(* CoDeSys 2.3.9.35 project: SISTEMA_2_SEMAFOROS.pro *)
(* Author: Franklin *)
(* Libraries: SysLibTargetVisu.lib 26.11.08 09:50:36, Standard.lib 26.11.08 09:46:20, Iecsfc.lib 26.11.08 09:46:14, DU35x.lib 26.11.09 14:36:14, SYSLIBCALLBACK.LIB 26.11.08 09:50:38 *)

(* PLC configuration (modules and I/O channels)
PLC Configuration [Root] node -1, in %IB0 out %QB0
  Communication [Comunica] node 0, in %IB0 out %QB0
    COM1 [COM1] node 0, in %IB0 out %QB0 {BaudRate = 115200; Paridade = No Parity; StopBits = 1 Stop Bit; Modem = Without RTS/CTS; Delay = 5}
      MToolIEC [Codesys] node 0, in %IB0 out %QB0
    COM2 [COM2] node 1, in %IB0 out %QB0 {BaudRate = 115200; Paridade = No Parity; StopBits = 1 Stop Bit; Modem = Without RTS/CTS; Delay = 5}
      Disable [Desabilitado485] node 0, in %IB0 out %QB0
  Bus [Barramento] node 1, in %IB0 out %QB0
    Inputs [Entradas] node 0, in %IB0 out %QB0
      Digital Inputs 0 [Entradas0] node 0, in %IW0 out %QB0
        I00 AT %IX0.0 [BitInput] I0.0
        I01 AT %IX0.1 [BitInput] I0.1
        I02 AT %IX0.2 [BitInput] I0.2
        I03 AT %IX0.3 [BitInput] I0.3
        I04 AT %IX0.4 [BitInput] I0.4
        I05 AT %IX0.5 [BitInput] I0.5
        I06 AT %IX0.6 [BitInput] I0.6
        I07 AT %IX0.7 [BitInput] I0.7
        I08 AT %IX0.8 [BitInput] I0.8
      Digital Inputs 1 [Entradas1] node 0, in %IW1 out %QB0
        I10 AT %IX1.0 [BitInput] I1.0
        I11 AT %IX1.1 [BitInput] I1.1
        I12 AT %IX1.2 [BitInput] I1.2
        I13 AT %IX1.3 [BitInput] I1.3
        I14 AT %IX1.4 [BitInput] I1.4
        I15 AT %IX1.5 [BitInput] I1.5
        I16 AT %IX1.6 [BitInput] I1.6
        I17 AT %IX1.7 [BitInput] I1.7
        I18 AT %IX1.8 [BitInput] I1.8
      Digital Inputs 2 [Entradas2] node 0, in %IW2 out %QB0
        I20 AT %IX2.0 [BitInput] I2.0
        I21 AT %IX2.1 [BitInput] I2.1
      Analog Inputs [EntradaAnalogica] node 0, in %IW4 out %QB0
        AI0 AT %IW4 [WordInput] AI0 {TipoAnalogica = Channel Disable; FiltroAnalogica = Filter 0 - AI=2ms  / AV=90ms; FundoEscala = 0}
        AI1 AT %IW5 [WordInput] AI1 {TipoAnalogica = Channel Disable; FiltroAnalogica = Filter 0 - AI=2ms  / AV=90ms; FundoEscala = 0}
        AI2 AT %IW6 [WordInput] AI2 {TipoAnalogica = Channel Disable; FiltroAnalogica = Filter 0 - AI=2ms  / AV=90ms; FundoEscala = 0}
        AI3 AT %IW7 [WordInput] AI3 {TipoAnalogica = Channel Disable; FiltroAnalogica = Filter 0 - AI=2ms  / AV=90ms; FundoEscala = 0}
      Fast Inputs [EntradasRapidas] node 1, in %IB16 out %QB0
        Block 0 [Bloco0] node 0, in %IB16 out %QB0
          Disable [DesabilitadoBloco0] node 0, in %IB16 out %QB0
        Block 1 [Bloco1] node 1, in %IB16 out %QB0
          Disable [DesabilitadoBloco1] node 0, in %IB16 out %QB0
        Configurable Input Block 0 [EntradaConfiBloco0] node 2, in %IB16 out %QB0
          Counter 0 [EntradaConfContador0] node 0, in %IB16 out %QB0 {EntradaConfiguravelContador = Disable}
        Configurable Input Block 1 [EntradaConfiBloco1] node 3, in %IB16 out %QB0
          Counter 2 [EntradaConfContador2] node 0, in %IB16 out %QB0 {EntradaConfiguravelContador = Disable}
    Outputs [Saidas] node 1, in %IB13 out %QB0
      Digital Outputs 0 [Saidas0] node 0, in %IW0 out %QW0
        Q00 AT %QX0.0 [BitOutput] Q0.0
        Q01 AT %QX0.1 [BitOutput] Q0.1
        Q02 AT %QX0.2 [BitOutput] Q0.2
        Q03 AT %QX0.3 [BitOutput] Q0.3
        Q04 AT %QX0.4 [BitOutput] Q0.4
        Q05 AT %QX0.5 [BitOutput] Q0.5
        Q06 AT %QX0.6 [BitOutput] Q0.6
        Q07 AT %QX0.7 [BitOutput] Q0.7
      Digital Outputs 1 [Saidas1] node 0, in %IW0 out %QW1
        Q10 AT %QX1.0 [BitOutput] Q1.0
        Q11 AT %QX1.1 [BitOutput] Q1.1
        Q12 AT %QX1.2 [BitOutput] Q1.2
        Q13 AT %QX1.3 [BitOutput] Q1.3
        Q14 AT %QX1.4 [BitOutput] Q1.4
        Q15 AT %QX1.5 [BitOutput] Q1.5
        Q16 AT %QX1.6 [BitOutput] Q1.6
        Q17 AT %QX1.7 [BitOutput] Q1.7
      Analog Outputs [SaidaAnalogica] node 0, in %IW0 out %QW3
        AO0 AT %QW3 [WordOutput] AO0 {TipoAnalogica = Channel Disable; FundoEscala = 0}
        AO1 AT %QW4 [WordOutput] AO1 {TipoAnalogica = Channel Disable; FundoEscala = 0}
      Fast Outputs [SaidasRapidas] node 1, in %IB0 out %QB10
        Fast Output 0 Disable [DesabilitadoF0] node 0, in %IB0 out %QB10
        Fast Output 1 Disable [DesabilitadoF1] node 1, in %IB0 out %QB10
      Counter Output [SaidasContador] node 2, in %IB0 out %QB10
        Block 0 Output Disable [DesabilitadoSaidaBloco0] node 0, in %IB0 out %QB10
        Block 1 Output Disable [DesabilitadoSaidaBloco1] node 1, in %IB0 out %QB10
  External Events [Eventos] node 2, in %IB13 out %QB6
    Timer Event [TimerEvent] node 0, in %IB13 out %QB6 {Intervalo = 10}
*)

(* POU PLC_PRG, LD *)
PROGRAM PLC_PRG
(*
	 autor; franklin
	 descricao: codigo estruturado com base em um autômato finito determinísco (AFD) para controle de maquina de estados finita
*)

VAR
	botao AT %IX0.0: BOOL;
	S0 AT %MX0.0: BOOL;
	T1: TON;
	A_VERDE AT %QX1.2: BOOL;
	B_VERMELHO AT %QX1.3: BOOL;
	S1 AT %MX0.1: BOOL;
	botao_pulso: R_TRIG;
	A_AMARELO AT %QX1.1: BOOL;
	T2: TON;
	S2 AT %MX0.2: BOOL;
	B_VERDE AT %QX1.5: BOOL;
	S3 AT %MX0.3: BOOL;
	A_VERMELHO AT %QX1.0: BOOL;
	B_AMARELO AT %QX1.4: BOOL;
	T3: TON;
	T4: TON;
END_VAR
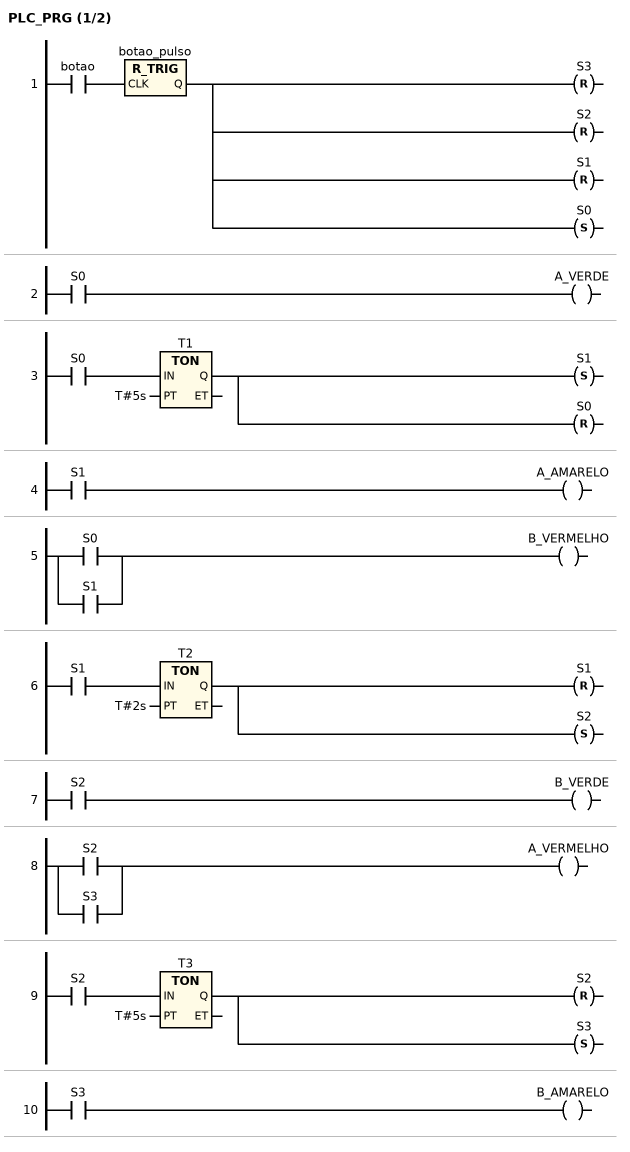
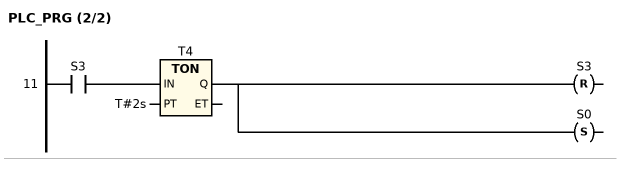
_LD_ (* Ladder Diagram *)
NETWORK 1
	[botao] - botao_pulso:R_TRIG(CLK: *) --- (R S3) (R S2) (R S1) (S S0)
NETWORK 2
	[S0] --- (A_VERDE)
NETWORK 3
	[S0] - T1:TON(IN: *, PT: T#5s) --- (S S1) (R S0)
NETWORK 4
	[S1] --- (A_AMARELO)
NETWORK 5
	{ [S0] | [S1] } --- (B_VERMELHO)
NETWORK 6
	[S1] - T2:TON(IN: *, PT: T#2s) --- (R S1) (S S2)
NETWORK 7
	[S2] --- (B_VERDE)
NETWORK 8
	{ [S2] | [S3] } --- (A_VERMELHO)
NETWORK 9
	[S2] - T3:TON(IN: *, PT: T#5s) --- (R S2) (S S3)
NETWORK 10
	[S3] --- (B_AMARELO)
NETWORK 11
	[S3] - T4:TON(IN: *, PT: T#2s) --- (R S3) (S S0)
_END_LD_
(* the same logic as Structured Text *)
(* Network 1 *)
botao_pulso(CLK := botao);
IF botao_pulso.Q THEN S3 := FALSE; S2 := FALSE; S1 := FALSE; S0 := TRUE; END_IF;
(* Network 2 *)
A_VERDE := S0;
(* Network 3 *)
T1(IN := S0, PT := T#5s);
IF T1.Q THEN S1 := TRUE; S0 := FALSE; END_IF;
(* Network 4 *)
A_AMARELO := S1;
(* Network 5 *)
B_VERMELHO := S0 OR S1;
(* Network 6 *)
T2(IN := S1, PT := T#2s);
IF T2.Q THEN S1 := FALSE; S2 := TRUE; END_IF;
(* Network 7 *)
B_VERDE := S2;
(* Network 8 *)
A_VERMELHO := S2 OR S3;
(* Network 9 *)
T3(IN := S2, PT := T#5s);
IF T3.Q THEN S2 := FALSE; S3 := TRUE; END_IF;
(* Network 10 *)
B_AMARELO := S3;
(* Network 11 *)
T4(IN := S3, PT := T#2s);
IF T4.Q THEN S3 := FALSE; S0 := TRUE; END_IF;
END_PROGRAM

(* Visualisation visualizacao1
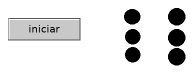
button at (14,13)-(86,35): text "iniciar"; toggles PLC_PRG.botao
ellipse at (131,42)-(146,57): alarm colour if PLC_PRG.A_VERDE
ellipse at (174,3)-(191,20): alarm colour if PLC_PRG.B_VERMELHO
ellipse at (131,24)-(146,39): alarm colour if PLC_PRG.A_AMARELO
ellipse at (130,4)-(146,19): alarm colour if PLC_PRG.A_VERMELHO
ellipse at (174,24)-(191,41): alarm colour if PLC_PRG.B_AMARELO
ellipse at (174,43)-(191,60): alarm colour if PLC_PRG.B_VERDE
*)
